{attribute addProperty BoxType "EL5101-0011-0016"}
{attribute addProperty Id "StatusAT %I*Status_23434B14162"}
{attribute addProperty CRC "1209836298"}
{attribute addProperty SizeInBites "16"}
{attribute addProperty SizeInBytes "2"}
TYPE ENC_Status_481CA30A :
STRUCT
	{attribute addProperty Name "Status"}
	Status AT %I* : Status_23434B14;
END_STRUCT
END_TYPE

(* stored: Version 1.2.0.0, ProductVersion 3.1.4024.9
   DUT ENC_Status_481CA30A: Id {bfe02b0c-f881-4aa2-9fbc-4841b35f1c46} *)
